TYPE ST_LinCoord_XYZ EXTENDS ST_LinCoord_XY :
STRUCT
	z	: REAL;	// [mm]
END_STRUCT
END_TYPE

(* stored: Version 1.1.0.1, ProductVersion 3.1.4026.18
   DUT ST_LinCoord_XYZ: Id {d135f31e-062e-41c0-854e-e50035b28398} *)
